{attribute 'qualified_only'}
VAR_GLOBAL CONSTANT
	test : BOOL := true;
END_VAR

(* stored: Version 1.1.0.1, ProductVersion 3.1.4024.12
   GVL Param: Id {270cee16-a6a4-46f1-a94a-b1b8e1a788dd}, ParameterList True *)
